FUNCTION TorrToMbar : REAL
VAR_INPUT
    pressure : REAL; // Torr
END_VAR

TorrToMbar := pressure * 1.3332236842;

END_FUNCTION

(* stored: Version 1.1.0.1, ProductVersion 3.1.4024.4
   POU TorrToMbar: Id {72443386-98ce-4f63-9f37-5583adb7777c}, SpecialFunc None *)
